PROGRAM PRG_Subscription
VAR
END_VAR

END_PROGRAM

(* stored: Version 1.1.0.1, ProductVersion 3.1.4024.9
   POU PRG_Subscription: Id {566e87ad-2ff3-47bb-b7ad-b791e069422f}, SpecialFunc None *)
